(* CODESYS project IoDrvTemplateIecDriverTest.project
   Title: IoDrvTemplate
   Version: 3.0.0.0
   Author: 3S - Smart Software Solutions GmbH
   Company: MyCompany

Project tree, tasks and I/O mapping:
  CODESYS_Control : CODESYS Control Win V3, 3S - Smart Software Solutions GmbH, version 3.5.14.10
    application Application
      libraries: CmpSupervisor, 3.5.11.0 (System)
      task T1 (cyclic, interval t#20ms, priority 1) calls Main
      task T2 (cyclic, interval t#20ms, priority 1) calls POU
      global variables GVL
      program Main [ST]
      program POU [ST]
    MyCard_IecDriver : MyCard_IecDriver, MyCompany, version 3.5.15.0
        input  Application.Main.dwIn1 : DWORD  // in1
        input  Application.Main.bitIn2 : BOOL  // in2.Bit1
        input  Application.POU.bitIn3 : BOOL  // in2.Bit3
        output Application.Main.dwOut1 : DWORD  // out1
        output Application.Main.bitOut2 : BOOL  // out2.Bit1
        output Application.POU.bitOut3 : BOOL  // out2.Bit3
        unmapped channels: in2, out2
*)

// CODESYS_Control/Application/GVL
VAR_GLOBAL RETAIN
	 B : DWORD;
END_VAR

// CODESYS_Control/Application/Main
PROGRAM Main
VAR
	A : DWORD;
	dwTest : DWORD;
	bEndlessLoop: BOOL;	// This is to test the behaviour of the outputs in software watchdog situations
	
	dwOut1 : DWORD;
	dwIn1 : DWORD;
	
	bitOut2 : BOOL;
	bitIn2 : BOOL;
	i : INT;
	
	(* reconfiguration test code for CAA Device Diagnosis *)
	Reconfig : DED.Reconfigure;	
	xEnableDevice : BOOL;
	xDisableWatchdog : BOOL;
	
	result : TPL.RTS_IEC_RESULT;
	ppIBase : POINTER TO POINTER TO BYTE;
	IBase : TPL.RTS_IEC_HANDLE;
	hOperation : TPL.RTS_IEC_HANDLE;
	pEntry : POINTER TO SupervisorEntry;
END_VAR

B := B + 1;

dwOut1 := dwIn1 - 1;

bitOut2 := bitIn2;

WHILE bEndlessLoop DO
	A := A + 1;
END_WHILE

B := B + 1;

// Reconfiguration test code for CAA Device Diagnosis to enable the IO-module dynamic
MyCard_IecDriver.Enable := xEnableDevice;
Reconfig(itfNode := MyCard_IECDriver);

IF xDisableWatchdog THEN
	xDisableWatchdog := FALSE;

	// Get IBase from out testdriver 
	ppIBase := MyCard_IecDriver.QueryInterface(TPL.ITFID_IBase, ADR(result));
	IBase := ppIBase^;
	
	// Iterate over all supervisor entries and check for the 
	hOperation := SupervisorOperationGetFirst(ADR(result));
	WHILE hOperation <> TPL.RTS_INVALID_HANDLE DO
		pEntry := SupervisorOperationGetEntry(hOperation, ADR(result));
		// Check, if the instance handle is our IBase pointer
		IF ((pEntry^.flags AND CmpSupervisor.SupervisorFlags.RTS_SUPERVISOR_FLAG_WATCHDOG) <> 0 AND	pEntry^.instance.xIsIECInstance = TRUE AND pEntry^.instance.hInstance =  IBase) THEN
			// Disable watchdog of this IO-driver! 
			SupervisorOperationDisable(hOperation);
			EXIT;
		END_IF
		hOperation := SupervisorOperationGetNext(hOperation, ADR(result));
	END_WHILE
END_IF

END_PROGRAM

// CODESYS_Control/Application/POU
PROGRAM POU
VAR
	bitOut3 : BOOL;
	bitIn3 : BOOL;
END_VAR

bitOut3;
bitIn3;

END_PROGRAM
